PROGRAM MAIN
VAR
	i :INT;
	m_Fbi_Soldering:FB_Soldering;
END_VAR

m_Fbi_Soldering.InStart:=SolderingStart;	
m_fbi_Soldering();

END_PROGRAM

(* stored: Version 1.1.0.1, ProductVersion 3.1.0.36
   POU MAIN: Id {fee2d26b-a3db-42c5-95e3-eb371e6dea0b}, SpecialFunc None *)
